{attribute addProperty BoxType "EL5122-0000-0016"}
{attribute addProperty Id "ENC_Status_ChannelAT %I*ARRAY[0..3] OF ENC_Status_Channel_1DBB2AA2192240ENC_Control_ChannelAT %Q*ARRAY[0..2] OF ENC_Control_Channel_50CA5D6096120WcStateAT %I*WcState_98A4DF7520.250InfoDataAT %I*InfoData_BC63D37F80100"}
{attribute addProperty CRC "4190224116"}
{attribute addProperty SizeInBites "370"}
{attribute addProperty SizeInBytes "46.25"}
TYPE EL5122_D4BE45F5 :
STRUCT
	{attribute addProperty Name "ENC_Status_Channel"}
	ENC_Status_Channel : ARRAY[0..3] OF ENC_Status_Channel_1DBB2AA2;
	{attribute addProperty Name "ENC_Control_Channel"}
	ENC_Control_Channel : ARRAY[0..2] OF ENC_Control_Channel_50CA5D60;
	{attribute addProperty Name "WcState"}
	WcState : WcState_98A4DF75;
	{attribute addProperty Name "InfoData"}
	InfoData : InfoData_BC63D37F;
END_STRUCT
END_TYPE

(* stored: Version 1.2.0.0, ProductVersion 3.1.4024.9
   DUT EL5122_D4BE45F5: Id {867ee423-2b17-4f35-9d2e-f2201d581a28} *)
